// TIA Portal V17 export
// export: Created 2023-12-22T15:05:28.8568582Z, ExportSetting WithDefaults, DisplayName Totally Integrated Automation Portal, DisplayVersion V17, DisplayName TIA Portal Openness, DisplayVersion V17, DisplayName TIA Portal Version Control Interface, DisplayVersion V17, DisplayName STEP 7 Professional, DisplayVersion V17, DisplayName STEP 7 Safety, DisplayVersion V17, DisplayName WinCC Advanced, DisplayVersion V17
DATA_BLOCK "Pump_1_DB"   // DB600
VERSION : 0.1
// stored: AutoNumber false, DBAccessibleFromOPCUA true, InstanceOfName DRV_M_DA, InstanceOfType FB
"DRV_M_DA"
   // VAR_INPUT
   //    All_Block : Bool;
   // END_VAR
   // VAR_IN_OUT
   //    FB_QF : Bool;
   //    FB_KM : Bool;
   //    S_Alarm : Bool;
   //    CMD_Run : Bool;
   // END_VAR
   // VAR RETAIN
   //    CMD : "CMD";
   //    Mode : Int;
   //    Status : Int;
   //    Use : Struct
   //       QF { S7_SetPoint := 'True'} : Bool := FALSE;
   //       KM { S7_SetPoint := 'True'} : Bool := TRUE;
   //       OpTime { S7_SetPoint := 'True'} : Bool := TRUE;
   //       Analog { S7_SetPoint := 'True'} : Bool := TRUE;
   //       Local_Keys : Bool;
   //    END_STRUCT;
   //    FB : Struct
   //       QF : Bool;
   //       KM : Bool;
   //       Local_Start : Bool;
   //       Local_Stop : Bool;
   //    END_STRUCT;
   //    ON : Bool;
   //    OFF : Bool;
   //    Tx { S7_SetPoint := 'True'} : Array[0..3] of "Time_S";
   //    Inv : Struct
   //       CMD { S7_SetPoint := 'True'} : Bool := FALSE;
   //       QF { S7_SetPoint := 'True'} : Bool := FALSE;
   //       KM { S7_SetPoint := 'True'} : Bool := FALSE;
   //    END_STRUCT;
   //    Alarm : Struct
   //       Block : Bool;
   //       QF : Bool;
   //       Start : Bool;
   //       Stop : Bool;
   //       Termo : Bool;
   //       Alarm : Bool;
   //       Safety : Bool;
   //       OpTime : Bool;
   //    END_STRUCT;
   //    Alarms : Word;
   //    Events : Word;
   //    pos : Array[0..15] of Bool;
   //    OpTime_h : DInt;
   //    OpTime_s { S7_SetPoint := 'True'} : DInt := 247244;
   //    OpTime_SP { S7_SetPoint := 'True'} : DInt := 2160;
   //    OpTime_Now_h : DInt;
   //    OpTime_Now_s { S7_SetPoint := 'True'} : DInt := 247244;
   //    CodeID { S7_SetPoint := 'True'} : Int := 0;
   //    Indirect : Struct
   //       FB_QF { S7_SetPoint := 'True'} : Bool := TRUE;
   //       FB_KM { S7_SetPoint := 'True'} : Bool := TRUE;
   //       CMD { S7_SetPoint := 'True'} : Bool := TRUE;
   //    END_STRUCT;
   //    Indirect_BYTE : Struct
   //       FB_QF { S7_SetPoint := 'True'} : Int := 0;
   //       FB_KM { S7_SetPoint := 'True'} : Int := 0;
   //       CMD { S7_SetPoint := 'True'} : Int := 0;
   //    END_STRUCT;
   //    Indirect_BIT : Struct
   //       FB_QF { S7_SetPoint := 'True'} : Int := 4;
   //       FB_KM { S7_SetPoint := 'True'} : Int := 3;
   //       CMD { S7_SetPoint := 'True'} : Int := 2;
   //    END_STRUCT;
   //    SP_A : Real;
   //    SP_M : Real;
   //    ADDR { S7_SetPoint := 'True'} : Int := 256;
   //    Converter { S7_SetPoint := 'True'} : "Converter";
   //    VmA : Real;
   //    Output_Type { S7_SetPoint := 'True'} : Int := 0;
   //    "Type" { S7_SetPoint := 'True'} : Int := 3;
   //    Slow { S7_SetPoint := 'True'} : "Slow";
   //    Time_DTL { S7_SetPoint := 'True'} : DTL := DTL#2012-01-01-20:29:19.377950;
   // END_VAR
BEGIN
   Tx[0].SP := 2;
   Tx[1].SP := 5;
   Tx[2].SP := 15;
   Tx[3].SP := 2;
   Converter.Lim_High := FALSE;
   Converter.Lim_Low := FALSE;
   Converter.Inverse := FALSE;
   Converter.Min_In := 0.0;
   Converter.Min_Out := 0.0;
   Converter.Max_In := 200.0;
   Converter.Max_Out := 27648.0;
   Slow.Use_Up := FALSE;
   Slow.Use_Down := FALSE;
   Slow.Step_Up := 0.125;
   Slow.Step_Down := 0.125;
   Slow.T_Up.SP := 1.0;
   Slow.T_Up.One := 0.1;
   Slow.T_Down.SP := 1.0;
   Slow.T_Down.One := 0.1;
END_DATA_BLOCK
